// TIA Portal V18 export
DATA_BLOCK "SS1_CPU1215_DI_Vars"   // DB11013
{ S7_Optimized_Access := 'FALSE' }
VERSION : 0.1
// stored: AutoNumber false, DBAccessibleFromOPCUA true, IsOnlyStoredInLoadMemory false, IsWriteProtectedInAS false
   VAR
      DI1 : "UDT_DIadv";
      DI2 : "UDT_DIadv";
      DI3 : "UDT_DIadv";
      DI4 : "UDT_DIadv";
      DI5 : "UDT_DIadv";
      DI6 : "UDT_DIadv";
      DI7 { S7_SetPoint := 'True'} : "UDT_DIadv";
      DI8 { S7_SetPoint := 'True'} : "UDT_DIadv";
      DI9 { S7_SetPoint := 'True'} : "UDT_DIadv";
      DI10 { S7_SetPoint := 'True'} : "UDT_DIadv";
      DI11 { S7_SetPoint := 'True'} : "UDT_DIadv";
      DI12 { S7_SetPoint := 'True'} : "UDT_DIadv";
      DI13 { S7_SetPoint := 'True'} : "UDT_DIadv";
      DI14 { S7_SetPoint := 'True'} : "UDT_DIadv";
   END_VAR
BEGIN
   DI1.cFuncSystemID := 3;
   DI1.cFuncVar := 19;
   DI2.cFuncSystemID := 3;
   DI2.cFuncVar := 8;
   DI3.cFuncSystemID := 3;
   DI3.cFuncVar := 9;
   DI4.cFuncSystemID := 3;
   DI4.cFuncVar := 20;
   DI5.cFuncSystemID := 3;
   DI5.cFuncVar := 7;
   DI6.cFuncSystemID := 3;
   DI6.cFuncVar := 21;
   DI8.cFuncSystemID := 10;
   DI8.cFuncVar := 41;
   DI9.cFuncSystemID := 10;
   DI9.cFuncVar := 43;
   DI10.cFuncSystemID := 3;
   DI10.cFuncVar := 16;
   DI11.cFuncSystemID := 3;
   DI11.cFuncVar := 18;
   DI12.cFuncSystemID := 10;
   DI12.cFuncVar := 29;
   DI13.cFuncSystemID := 10;
   DI13.cFuncVar := 28;
END_DATA_BLOCK
